VAR 
	i :INT;
END_VAR
// enable/disenable joint5
IF i_setupArm.jnt5AdjustDir = 0 THEN
	m_jntEnableFlag[5] := 0;
	m_cmdJntPos[5]:=i_setupArm.curJntPos[5];
	m_jnt5EnableTime:=0;
	m_cmdJntVel[5]:=0;
	RETURN;
ELSE
	m_jntEnableFlag[5] := 1;
	m_jnt5EnableTime := m_jnt5EnableTime + g_setupArmCtrlCycleTime;
END_IF

// update command position
IF m_jnt5EnableTime>m_jnt5AdjustWaitTime THEN
	m_cmdJntVel[5]:=m_cmdJntVel[5] + i_setupArm.jnt5AdjustDir * m_jnt5MaxAdjustAcc * g_setupArmCtrlCycleTime;
	m_cmdJntVel[5]:=LIMIT(-m_jnt5MaxAdjustVel, m_cmdJntVel[5], m_jnt5MaxAdjustVel);
	
	// joint limit
	IF (m_cmdJntPos[5] > GVL_SetupMotorParameters.g_maxJntPos[i_setupArm.armIdx, 5] AND m_cmdJntVel[5]>0) OR (m_cmdJntPos[5] < GVL_SetupMotorParameters.g_minJntPos[i_setupArm.armIdx, 5] AND m_cmdJntVel[5]<0)  THEN
		m_cmdJntVel[5] := 0;
	END_IF
	
	m_cmdJntPos[5]:= m_cmdJntPos[5] + m_cmdJntVel[5] * g_setupArmCtrlCycleTime;
END_IF
END_METHOD

// override this function in each exact controller
METHOD PROTECTED calcCmdJntTrq : BOOL
VAR_IN_OUT CONSTANT
	i_setupArm	:FB_SetupArm;
END_VAR
VAR
	i:INT;
	vel :LREAL;
	scale:LREAL;
	ratio:LREAL;
END_VAR
// set joint torque to zero in default
m_cmdJntTrq := g_zeroVec5d;

//enable/diable  joint1-4
IF NOT(i_setupArm.manualAdjustOn) THEN
	FOR i:=1 TO 4 DO
		m_jntEnableFlag[i] := 0;
		m_jntOPMode[i]:=DriverOPMode_Pos;
	END_FOR
	RETURN;
ELSE
	FOR i:=1 TO 4 DO
		m_jntEnableFlag[i] := 1;
		m_jntOPMode[i]:=DriverOPMode_Trq;
		m_cmdJntPos[i] := i_setupArm.curJntPos[i];
	END_FOR
END_IF

// friction scale
vel:=ABS(i_setupArm.curJntVel[3]);
IF vel < m_jnt3FrictionCompVelLow THEN
	m_frictionScale := m_frictionScaleLow * vel/m_jnt3FrictionCompVelLow ;
ELSIF  vel > m_jnt3FrictionCompVelLow AND vel  < m_jnt3FrictionCompVelMiddle THEN
	ratio:= (vel-m_jnt3FrictionCompVelLow)/(m_jnt3FrictionCompVelMiddle-m_jnt3FrictionCompVelLow);
	m_frictionScale :=m_frictionScaleLow+ratio * (m_frictionScaleMiddle-m_frictionScaleLow);
ELSIF  vel > m_jnt3FrictionCompVelMiddle AND vel  < m_jnt3FrictionCompVelHigh THEN
	ratio:= (vel-m_jnt3FrictionCompVelMiddle)/(m_jnt3FrictionCompVelHigh-m_jnt3FrictionCompVelMiddle);
	m_frictionScale :=m_frictionScaleMiddle+ratio * (m_frictionScaleHigh-m_frictionScaleMiddle);
ELSIF  vel > m_jnt3FrictionCompVelHigh THEN
	m_frictionScale := m_frictionScaleHigh;
END_IF

// add friction compensation
m_frictionScale := LIMIT(0, m_frictionScale, 1);
m_cmdJntTrq[3]:= m_frictionScale * sign(i_setupArm.curJntVel[3])*jnt3Friction(i_setupArm.armIdx, i_setupArm.curJntPos[3]);
END_METHOD

METHOD PUBLIC init : BOOL
VAR_IN_OUT CONSTANT
	i_setupArm	:FB_SetupArm;
END_VAR
VAR_IN_OUT 
	r_setupArmCtrlCmd :ST_SetupArmCtrlCmds;
END_VAR
SUPER^.Init(i_setupArm,r_setupArmCtrlCmd);
m_jnt5EnableTime :=0;
END_METHOD

METHOD PROTECTED jnt3Friction : Lreal
VAR_INPUT
	i_armIdx:INT;
	i_jnt3Pos :LREAL;
END_VAR

VAR
	q:LREAL;
END_VAR
q := LIMIT(GVL_SetupArmDynamics.g_setupJnt3GravityPosRange[i_armIdx,1], i_jnt3Pos, GVL_SetupArmDynamics.g_setupJnt3GravityPosRange[i_armIdx,2]);
jnt3Friction:=GVL_SetupArmDynamics.g_setupJnt3FrictionParams[i_armIdx,1]*EXPT(q,3)+GVL_SetupArmDynamics.g_setupJnt3FrictionParams[i_armIdx,2]*EXPT(q,2)+
				GVL_SetupArmDynamics.g_setupJnt3FrictionParams[i_armIdx,3]*q+GVL_SetupArmDynamics.g_setupJnt3FrictionParams[i_armIdx,4];
END_METHOD

END_FUNCTION_BLOCK

// ---- FBs_SlaveControllers/FB_SlaveCtrlInstruInvasion.TcPOU
// Brief: Slave Arm Adjust
FUNCTION_BLOCK PUBLIC FB_SlaveCtrlInstruInvasion EXTENDS FB_SlaveArmCtrlBase
VAR_INPUT
END_VAR
VAR_OUTPUT
END_VAR
VAR
	// invasion buffer
	m_instruInvasionDepthSafetyBuffer :LREAL:= 0.01;
		
	// max damping when reaching invasion depth
	m_maxDamp :LREAL :=500;
	
	// current distance form target invasion depth 
	m_invasionDis :LREAL :=0;
	
	// distance threshold from target depth to start enable damp
	m_dampDisThres :LREAL :=0.03;
	
END_VAR

// override this function in each exact controller
METHOD PROTECTED calcCmdJntPos : BOOL
VAR_IN_OUT CONSTANT
	i_endoscopePose : ST_Frame;
	i_masterStatus :ST_MasterStatus;
	i_setupStatus: ST_SetupStatus;
	i_slaveArm :FB_SlaveArm;
END_VAR

VAR 
	curInstruDepth:LREAL;
END_VAR
m_cmdJntPos[3]:=i_slaveArm.curJntPos[3];
// compute current instrument depth
curInstruDepth := i_slaveArm.curJntPos[3]-i_slaveArm.instrument.kinematicParameters.m_rodLength-i_slaveArm.instrument.kinematicParameters.m_headLength
						- i_slaveArm.instrument.kinematicParameters.m_fingerLength-m_instruInvasionDepthSafetyBuffer;

m_invasionDis:=curInstruDepth-i_slaveArm.m_instruInvasionDepth;
						
m_isFinished := curInstruDepth<= i_slaveArm.m_instruInvasionDepth;
END_METHOD

// override this function in each exact controller
METHOD PROTECTED calcCmdJntTrq : BOOL
VAR_IN_OUT CONSTANT
	i_endoscopePose : ST_Frame;
	i_masterStatus :ST_MasterStatus;
	i_setupStatus: ST_SetupStatus;
	i_slaveArm :FB_SlaveArm;
END_VAR
VAR
	dampScale :lreal ;
END_VAR
// set joint torque to zero in default
m_cmdJntTrq := g_zeroVec8d;

dampScale  :=LIMIT(0, 1-m_invasionDis/m_dampDisThres,1);
m_cmdJntTrq[3]:= -dampScale * m_maxDamp * i_slaveArm.curJntVel[3];
END_METHOD

METHOD PUBLIC init : BOOL
VAR_IN_OUT CONSTANT
	i_slaveArm	:FB_SlaveArm;
END_VAR
VAR_IN_OUT 
	r_slaveArmCtrlCmd :ST_SlaveArmCtrlCmds;
END_VAR
// check if to hold the command joint position unchanged
m_holdLastCmds := checkToHoldLastCmds(i_slaveArm);

//init
SUPER^.Init(i_slaveArm,r_slaveArmCtrlCmd);
m_invasionDis:=m_dampDisThres;

// only joint 3 is allowed to be pushed
m_jntOPMode := g_slaveAllPosMode;
m_jntOPMode[3]:=DriverOPMode_Trq;

// update commands to arm
copyCmds(r_slaveArmCtrlCmd);
END_METHOD

END_FUNCTION_BLOCK

// ---- FBs_SlaveControllers/FB_SlaveCtrlInstruCali.TcPOU
// Brief: Mounting Instrument
FUNCTION_BLOCK PUBLIC FB_SlaveCtrlInstruCali EXTENDS FB_SlaveArmCtrlBase
VAR
	// mount motion planning
	m_jntOTG :ARRAY[1..8] OF FB_secOrdTrajFilter;
	m_instruMountVel :LREAL := 2*PI;
	m_instruMountAcc :LREAL := 4*PI;
	
	// 	cali status
	m_rollJntCaliStatus :INT := 0;
	m_pitchJntCaliStatus :INT := 0;
	m_yawJntCaliStatus :INT := 0;
	
	// flag if zero position is written to CoE
	m_zeroPosWritten :BOOL;
	
	// joint current threshold which indicate panel is buckled with instrument
	m_maxJntCurrent :LREAL := 100;
	
	// joint current threshold which indicate finger closed
	m_fingerCloseCurrent :LREAL := 50;
	
	// joint position at limits
	m_jntLimitPos1, m_jntLimitPos2, m_jntCaliPos :LREAL;
	m_jntLimitPos3, m_jntLimitPos4 :LREAL;

	// flag if joint is mounted
	m_jointMounted :ARRAY[1..8] OF BOOL := [5(FALSE)];
	
	// instrument mount motion range
	m_mountMotionAng :LREAL :=pi;
	
	// command mount motion
	m_targetMountPos :Vec8d;
	
	// instrument zero position
	m_instruZeroPosition :Vec5d;
	
END_VAR

// override this function in each exact controller
METHOD PROTECTED calcCmdJntPos : BOOL
VAR_IN_OUT CONSTANT
	i_endoscopePose : ST_Frame;
	i_masterStatus :ST_MasterStatus;
	i_setupStatus: ST_SetupStatus;
	i_slaveArm :FB_SlaveArm;
END_VAR

VAR 
	i :INT;
END_VAR
// retur directly if instrument/endoscope is not readed
IF NOT i_slaveArm.instrument.onChipData.m_InstruReadSucceed THEN
	m_rollJntCaliStatus :=0;
	m_pitchJntCaliStatus :=0;
	m_yawJntCaliStatus :=0;
	m_zeroPosWritten :=FALSE;
	FOR i:=4 TO 8 DO
		m_jointMounted[i]:=FALSE;
	END_FOR
	return;
END_IF

// write zero position to CoE
IF m_yawJntCaliStatus = -1 THEN
	IF   NOT m_zeroPosWritten THEN
		m_zeroPosWritten := i_slaveArm.instrument.writeZeroPosToChip(m_instruZeroPosition[1],m_instruZeroPosition[2],m_instruZeroPosition[3]);
	END_IF
	RETURN;
END_IF;

// move joint to zero position
IF m_rollJntCaliStatus <> -1 THEN
	rollJntCali(i_slaveArm);
ELSIF m_pitchJntCaliStatus <> -1 THEN
	pitchJntCali(i_slaveArm);
ELSIF m_yawJntCaliStatus <> -1 THEN
	IF  i_slaveArm.instrument.m_isSingleFinger THEN
		yawJntCali_finger(i_slaveArm);
	ELSE
		yawJntCali_gripper(i_slaveArm);
	END_IF

END_IF

IF m_yawJntCaliStatus = -1 THEN
	FOR  i:=1 TO  5 DO
		m_instruZeroPosition[i]:=i_slaveArm.linkSingle[i+3];
	END_FOR
END_IF
END_METHOD

METHOD PUBLIC init : BOOL
VAR_IN_OUT CONSTANT
	i_slaveArm	:FB_SlaveArm;
END_VAR
VAR_IN_OUT 
	r_slaveArmCtrlCmd :ST_SlaveArmCtrlCmds;
END_VAR

VAR
	i : INT;
END_VAR
// check if to hold the command joint position unchanged
m_holdLastCmds := checkToHoldLastCmds(i_slaveArm);

SUPER^.Init(i_slaveArm,r_slaveArmCtrlCmd);
m_jntOPMode[4] := DriverOPMode_PosTrq;
m_jntOPMode[5] := DriverOPMode_PosTrq;
m_jntOPMode[6] := DriverOPMode_PosTrq;
m_jntOPMode[7] := DriverOPMode_PosTrq;
m_jntOPMode[8] := DriverOPMode_PosTrq;

FOR i:=4 TO 8 DO
	m_targetMountPos[i]:=m_cmdJntPos[i];
	m_jntOTG[i].init(m_targetMountPos[i], 0,m_instruMountVel, m_instruMountAcc, g_slaveArmCtrlCycleTime);
	m_jointMounted[i]:=FALSE;
END_FOR

m_rollJntCaliStatus :=0;
m_pitchJntCaliStatus :=0;
m_yawJntCaliStatus :=0;
m_zeroPosWritten := false;

// update commands to arm
copyCmds(r_slaveArmCtrlCmd);
END_METHOD

METHOD pitchJntCali : BOOL
VAR_IN_OUT CONSTANT
	i_slaveArm :FB_SlaveArm;
END_VAR

VAR 
	i :INT;
	curJntPos :Vec8d;
	jntIdx :INT;
END_VAR
jntIdx:=6;
curJntPos := i_slaveArm.curJntPos;

CASE m_pitchJntCaliStatus OF
	// rotate clockwise
	0:
		m_targetMountPos[jntIdx]:=curJntPos[jntIdx]+m_mountMotionAng;
	
		//buckle joint
		IF i_slaveArm.filtJntCurrent[jntIdx]> m_maxJntCurrent THEN 
			m_jntLimitPos1 := curJntPos[jntIdx];
			m_targetMountPos[jntIdx]:=curJntPos[jntIdx];
			m_jntOTG[jntIdx].init(m_targetMountPos[jntIdx], 0,m_instruMountVel, m_instruMountAcc, g_slaveArmCtrlCycleTime);
			m_pitchJntCaliStatus := 1;
		END_IF
		
	// rotate anticlockwise
	1:
		m_targetMountPos[jntIdx]:=curJntPos[jntIdx]-m_mountMotionAng;
	
		//buckle  joint
		IF i_slaveArm.filtJntCurrent[jntIdx]<- m_maxJntCurrent THEN 
			m_jntLimitPos2 := curJntPos[jntIdx];
			m_targetMountPos[jntIdx]:=curJntPos[jntIdx];
			m_jntOTG[jntIdx].init(m_targetMountPos[jntIdx], 0,m_instruMountVel, m_instruMountAcc, g_slaveArmCtrlCycleTime);
			m_pitchJntCaliStatus := 2;
		END_IF
	
	2:// calculate center/calibarted position
		m_targetMountPos[jntIdx] :=  (m_jntLimitPos1 + m_jntLimitPos2)/2;
		m_pitchJntCaliStatus := 3;

	3:
		IF ABS(m_targetMountPos[jntIdx]-curJntPos[jntIdx]) <GVL_SlaveControlParameters.g_jntCtrlAngTolHigh  THEN
			m_pitchJntCaliStatus := -1;
		END_IF
		
END_CASE

// traj plan
m_jntOTG[jntIdx].run(m_targetMountPos[jntIdx],0.0, o_cmdAcc=>m_cmdJntAcc[jntIdx],o_cmdVel=>m_cmdJntVel[jntIdx],o_cmdPos=>m_cmdJntPos[jntIdx]);
END_METHOD

METHOD rollJntCali : BOOL
VAR_IN_OUT CONSTANT
	i_slaveArm :FB_SlaveArm;
END_VAR

VAR 
	i :INT;
	curJntPos :Vec8d;
	jntIdx :INT;
END_VAR
jntIdx:=7;
curJntPos := i_slaveArm.curJntPos;

CASE m_rollJntCaliStatus OF
	// rotate clockwise
	0:
		m_targetMountPos[jntIdx]:=curJntPos[jntIdx]+m_mountMotionAng;
	
		//buckle  joint
		IF i_slaveArm.filtJntCurrent[jntIdx]> m_maxJntCurrent THEN 
			m_jntLimitPos1 := curJntPos[jntIdx];
			m_targetMountPos[jntIdx]:=curJntPos[jntIdx];
			m_jntOTG[jntIdx].init(m_targetMountPos[jntIdx], 0,m_instruMountVel, m_instruMountAcc, g_slaveArmCtrlCycleTime);
			m_rollJntCaliStatus := 1;
		END_IF
		
	// rotate anticlockwise
	1:
		m_targetMountPos[jntIdx]:=curJntPos[jntIdx]-m_mountMotionAng;
	
		//buckle  joint
		IF i_slaveArm.filtJntCurrent[jntIdx]<- m_maxJntCurrent THEN 
			m_jntLimitPos2 := curJntPos[jntIdx];
			m_targetMountPos[jntIdx]:=curJntPos[jntIdx];
			m_jntOTG[jntIdx].init(m_targetMountPos[jntIdx], 0,m_instruMountVel, m_instruMountAcc, g_slaveArmCtrlCycleTime);
			m_rollJntCaliStatus := 2;
		END_IF
	
	2:// calculate center/calibarted positio
		m_targetMountPos[jntIdx] :=  (m_jntLimitPos1 + m_jntLimitPos2)/2;
		m_rollJntCaliStatus := 3;

	3:
		IF ABS(m_targetMountPos[jntIdx]-curJntPos[jntIdx]) <GVL_SlaveControlParameters.g_jntCtrlAngTolHigh  THEN
			m_rollJntCaliStatus := -1;
		END_IF
		
END_CASE

// traj plan
m_jntOTG[jntIdx].run(m_targetMountPos[jntIdx],0.0, o_cmdAcc=>m_cmdJntAcc[jntIdx],o_cmdVel=>m_cmdJntVel[jntIdx],o_cmdPos=>m_cmdJntPos[jntIdx]);
END_METHOD

METHOD yawJntCali_finger : BOOL
VAR_IN_OUT CONSTANT
	i_slaveArm :FB_SlaveArm;
END_VAR

VAR 
	i :INT;
	curJntPos :Vec8d;
	jntIdx :INT;
END_VAR
jntIdx:=5;
curJntPos := i_slaveArm.curJntPos;

CASE m_yawJntCaliStatus OF
	// rotate clockwise
	0:
		m_targetMountPos[jntIdx]:=curJntPos[jntIdx]+m_mountMotionAng;
	
		//buckle  joint
		IF i_slaveArm.filtJntCurrent[jntIdx]> m_maxJntCurrent THEN 
			m_jntLimitPos1 := curJntPos[jntIdx];
			m_targetMountPos[jntIdx]:=curJntPos[jntIdx];
			m_jntOTG[jntIdx].init(m_targetMountPos[jntIdx], 0,m_instruMountVel, m_instruMountAcc, g_slaveArmCtrlCycleTime);
			m_yawJntCaliStatus := 1;
		END_IF
		
	// rotate anticlockwise
	1:
		m_targetMountPos[jntIdx]:=curJntPos[jntIdx]-m_mountMotionAng;
	
		//buckle  joint
		IF i_slaveArm.filtJntCurrent[jntIdx]<- m_maxJntCurrent THEN 
			m_jntLimitPos2 := curJntPos[jntIdx];
			m_targetMountPos[jntIdx]:=curJntPos[jntIdx];
			m_jntOTG[jntIdx].init(m_targetMountPos[jntIdx], 0,m_instruMountVel, m_instruMountAcc, g_slaveArmCtrlCycleTime);
			m_yawJntCaliStatus := 2;
		END_IF
	
	2:// calculate center/calibarted positio
		m_targetMountPos[jntIdx] :=  (m_jntLimitPos1 + m_jntLimitPos2)/2;
		m_yawJntCaliStatus := 3;

	3:
		IF ABS(m_targetMountPos[jntIdx]-curJntPos[jntIdx]) <GVL_SlaveControlParameters.g_jntCtrlAngTolHigh  THEN
			m_yawJntCaliStatus := -1;
		END_IF
		
END_CASE

// traj plan
m_jntOTG[jntIdx].run(m_targetMountPos[jntIdx],0.0, o_cmdAcc=>m_cmdJntAcc[jntIdx],o_cmdVel=>m_cmdJntVel[jntIdx],o_cmdPos=>m_cmdJntPos[jntIdx]);
END_METHOD

METHOD yawJntCali_gripper : BOOL
VAR_IN_OUT CONSTANT
	i_slaveArm :FB_SlaveArm;
END_VAR

VAR 
	i :INT;
	curJntPos :Vec8d;
	jntRange:LREAL;
	jntIdx :INT;
END_VAR
curJntPos := i_slaveArm.curJntPos;

CASE m_yawJntCaliStatus OF
	// roll clockwise
	0:
		//buckle panel with instrument
		// check if buckled 
		IF i_slaveArm.filtJntCurrent[4]<- m_maxJntCurrent THEN 
			m_jointMounted[4]:=TRUE;
			m_targetMountPos[4]:=curJntPos[4];
			m_jntOTG[4].init(m_targetMountPos[4], 0,m_instruMountVel, m_instruMountAcc, g_slaveArmCtrlCycleTime);
		END_IF
		IF i_slaveArm.filtJntCurrent[5]> m_maxJntCurrent THEN 
			m_jointMounted[5]:=TRUE;
			m_targetMountPos[5]:=curJntPos[5];
			m_jntOTG[5].init(m_targetMountPos[5], 0,m_instruMountVel, m_instruMountAcc, g_slaveArmCtrlCycleTime);
		END_IF
		
		// set target joint position
		IF FALSE = m_jointMounted[4] THEN
			m_targetMountPos[4]:=curJntPos[4]-m_mountMotionAng;
		END_IF
		IF FALSE = m_jointMounted[5] THEN
			m_targetMountPos[5]:=curJntPos[5]+m_mountMotionAng;
		END_IF

		IF m_jointMounted[4] AND m_jointMounted[5] THEN
			m_jntLimitPos1 := curJntPos[4];
			m_jntLimitPos2 := curJntPos[5];
			m_yawJntCaliStatus := 1;
			m_jointMounted[4]:=FALSE;
			m_jointMounted[5]:=FALSE;
		END_IF

	// roll anticlockwise
	1:
		IF i_slaveArm.filtJntCurrent[4]> m_maxJntCurrent THEN 
			m_jointMounted[4]:=TRUE;
			m_targetMountPos[4]:=curJntPos[4];
			m_jntOTG[4].init(m_targetMountPos[4], 0,m_instruMountVel, m_instruMountAcc, g_slaveArmCtrlCycleTime);
		END_IF
		IF i_slaveArm.filtJntCurrent[5]<- m_maxJntCurrent THEN 
			m_jointMounted[5]:=TRUE;
			m_targetMountPos[5]:=curJntPos[5];
			m_jntOTG[5].init(m_targetMountPos[5], 0,m_instruMountVel, m_instruMountAcc, g_slaveArmCtrlCycleTime);
		END_IF
		
		// set target joint position
		IF FALSE = m_jointMounted[4] THEN
			m_targetMountPos[4]:=curJntPos[4]+m_mountMotionAng;
		END_IF
		IF FALSE = m_jointMounted[5] THEN
			m_targetMountPos[5]:=curJntPos[5]-m_mountMotionAng;
		END_IF
		
		IF m_jointMounted[4] AND m_jointMounted[5] THEN
			m_jntLimitPos3 := curJntPos[4];
			m_jntLimitPos4 := curJntPos[5];
			m_yawJntCaliStatus :=2;
			m_jointMounted[4]:=FALSE;
			m_jointMounted[5]:=FALSE;
		END_IF
		
	2:// calculate center/calibarted position
		m_targetMountPos[4] := (m_jntLimitPos1 + m_jntLimitPos3)/2;
		m_targetMountPos[5] := (m_jntLimitPos2 + m_jntLimitPos4)/2;
		m_yawJntCaliStatus := 3;

	3:
		IF ABS(m_targetMountPos[4]-curJntPos[4]) <GVL_SlaveControlParameters.g_jntCtrlAngTolHigh  AND
			ABS(m_targetMountPos[5]-curJntPos[5]) <GVL_SlaveControlParameters.g_jntCtrlAngTolHigh  THEN
			m_yawJntCaliStatus := 4;
		END_IF
		
	// close finger
	4:
		//buckle panel with instrument
		FOR i:=4 TO 5 DO
			// check if buckled 
			IF i_slaveArm.filtJntCurrent[i]> m_fingerCloseCurrent THEN 
				m_jointMounted[i]:=TRUE;
				m_targetMountPos[i]:=curJntPos[i];
				m_jntOTG[i].init(m_targetMountPos[i], 0,m_instruMountVel, m_instruMountAcc, g_slaveArmCtrlCycleTime);
			END_IF
			
			// set target joint position
			IF FALSE = m_jointMounted[i] THEN
				m_targetMountPos[i]:=curJntPos[i]+m_mountMotionAng;
			END_IF
		END_FOR
		
		IF m_jointMounted[4] AND m_jointMounted[5] THEN
			m_yawJntCaliStatus := -1;
		END_IF
END_CASE

// traj plan
m_jntOTG[4].run(m_targetMountPos[4],0.0, o_cmdAcc=>m_cmdJntAcc[4],o_cmdVel=>m_cmdJntVel[4],o_cmdPos=>m_cmdJntPos[4]);
m_jntOTG[5].run(m_targetMountPos[5],0.0, o_cmdAcc=>m_cmdJntAcc[5],o_cmdVel=>m_cmdJntVel[5],o_cmdPos=>m_cmdJntPos[5]);
END_METHOD

END_FUNCTION_BLOCK

// ---- FBs_SlaveControllers/FB_SlaveCtrlError.TcPOU
// Brief: Slave Arm Error Hold
FUNCTION_BLOCK PUBLIC FB_SlaveCtrlError EXTENDS FB_SlaveArmCtrlBase
VAR_INPUT
END_VAR
VAR_OUTPUT
END_VAR
VAR
END_VAR

// override this function in each exact controller
METHOD PROTECTED calcCmdJntPos : BOOL
VAR_IN_OUT CONSTANT
	// endoscope pose in cart coordinate
	i_endoscopePose : ST_Frame;
	
	// master arm data
	i_masterStatus :ST_MasterStatus;
	
	// setup arm data
	i_setupStatus: ST_SetupStatus;
	
	// slave arm data
	i_slaveArm :FB_SlaveArm;
END_VAR
m_cmdJntPos := i_slaveArm.curJntPos;
END_METHOD

// override this function in each exact controller
// NOTICE: set joint control mode here, and do some initialization if needed
METHOD PUBLIC init : BOOL
VAR_IN_OUT CONSTANT
	i_slaveArm	:FB_SlaveArm;
END_VAR
VAR_IN_OUT 
	r_slaveArmCtrlCmd :ST_SlaveArmCtrlCmds;
END_VAR


VAR
	i:INT;
END_VAR
SUPER^.Init(i_slaveArm,r_slaveArmCtrlCmd);

// disable all joints
 m_jntEnableFlag :=g_zeroVec8i;
 
 // update commands to arm
copyCmds(r_slaveArmCtrlCmd);
END_METHOD

END_FUNCTION_BLOCK

// ---- FBs_SlaveControllers/FB_SlaveCtrlMountInstru.TcPOU
// Brief: Mounting Instrument
FUNCTION_BLOCK PUBLIC FB_SlaveCtrlMountInstru EXTENDS FB_SlaveArmCtrlBase
VAR
	// mount status
	m_instruMountStatus :INT := 0;
	m_scopeMountStatus :INT := 0;
	m_ultrasoundMountStatus :INT :=0 ;
	
	// flag if joint is mounted
	m_jointMounted :ARRAY[1..5] OF BOOL := [5(FALSE)];
	
	// instrument mount motion range
	m_mountMotionAng :Vec5d :=[5(pi)];
	
	// instrument mount direction
	m_mountDir :Vec5i :=[1, 1, 1, 1, 1];
	
	// mount motion planning
	m_jntOTG :ARRAY[1..5] OF FB_secOrdTrajFilter;
	m_instruMountVel :LREAL := 4*PI;
	m_instruMountAcc :LREAL := 8*PI;
	
	//Joint 4 half-range angle of instrument
	m_instruJnt4HalfRangeAng :LREAL := 323*g_deg2Rad;
	
	// joint current threshold which indicate panel is buckled with instrument
	m_maxJntCurrent :Vec5d := [150, 150, 150, 180, 180];
	
	// command mount motion
	m_targetMountPos :Vec8d;
	
	// instrument zero position
	m_instruZeroDeviation :Vec5d;
	
	//ultrasound knife Reduce the current rotation Angle  J3
	m_ultraKnifeRotaAngleJ3 :LREAL := 3*g_deg2Rad;
	
	// joint position error
	m_jntPosErr :Vec5d;
	
	// endoscope motion angle to original position
	m_scopeJnt4CenterMotionAng :LREAL :=175*g_deg2Rad;
	m_scopeJnt5CenterMotionAng :LREAL :=150*g_deg2Rad;
	
END_VAR

// override this function in each exact controller
METHOD PROTECTED calcCmdJntPos : BOOL
VAR_IN_OUT CONSTANT
	i_endoscopePose : ST_Frame;
	i_masterStatus :ST_MasterStatus;
	i_setupStatus: ST_SetupStatus;
	i_slaveArm :FB_SlaveArm;
END_VAR

VAR 
END_VAR
// return directly if instrument/endoscope is not readed
IF i_slaveArm.instrument.onChipData.m_Error THEN
	return;
END_IF

IF i_slaveArm.instrument.onChipData.m_InstruReadSucceed AND InstruType_endoscope = i_slaveArm.instrument.m_instruType THEN
	mountEndoscope(i_slaveArm);
ELSIF i_slaveArm.instrument.onChipData.m_InstruReadSucceed AND InstruType_UltrasoundKnife = i_slaveArm.instrument.m_instruType THEN
	mountUltraKnife(i_slaveArm);
ELSE
	mountInstrument(i_slaveArm);
END_IF
END_METHOD

METHOD PUBLIC init : BOOL
VAR_IN_OUT CONSTANT
	i_slaveArm	:FB_SlaveArm;
END_VAR
VAR_IN_OUT 
	r_slaveArmCtrlCmd :ST_SlaveArmCtrlCmds;
END_VAR

VAR
	i : INT;
END_VAR
// check if to hold the command joint position unchanged
m_holdLastCmds := checkToHoldLastCmds(i_slaveArm);

SUPER^.Init(i_slaveArm,r_slaveArmCtrlCmd);
m_jntOPMode[4] := DriverOPMode_PosTrq;
m_jntOPMode[5] := DriverOPMode_PosTrq;
m_jntOPMode[6] := DriverOPMode_PosTrq;
m_jntOPMode[7] := DriverOPMode_PosTrq;
m_jntOPMode[8] := DriverOPMode_PosTrq;

FOR i:=1 TO 5 DO
	m_targetMountPos[i+3]:=m_cmdJntPos[i+3];
	m_jntOTG[i].init(m_targetMountPos[i+3], 0,m_instruMountVel, m_instruMountAcc, g_slaveArmCtrlCycleTime);
	m_jointMounted[i]:=FALSE;
END_FOR

m_instruMountStatus:=0;
m_scopeMountStatus:=0;
m_ultrasoundMountStatus:=0;

// update commands to arm
copyCmds(r_slaveArmCtrlCmd);
END_METHOD

METHOD mountEndoscope : BOOL
VAR_IN_OUT CONSTANT
	i_slaveArm :FB_SlaveArm;
END_VAR

VAR 
	i :INT;
	curJntPos :Vec8d;
END_VAR
curJntPos := i_slaveArm.curJntPos;

CASE m_scopeMountStatus OF
	//fix scope lock joint(joint 7)
	0:
		// other joints stay still
		FOR i:=1 TO 3 DO
			m_jointMounted[i] := TRUE;
			m_targetMountPos[i+3]:=curJntPos[i+3];
			m_jntOTG[i].init(m_targetMountPos[i+3], 0,m_instruMountVel, m_instruMountAcc, g_slaveArmCtrlCycleTime);
		END_FOR
	
		// check if buckled
		m_jointMounted[4]:=FALSE; 
		m_jointMounted[5]:=FALSE; 
		IF ABS(i_slaveArm.filtJntCurrent[7])> m_maxJntCurrent[4] THEN 
			m_jointMounted[4]:=TRUE;
			m_targetMountPos[7]:=curJntPos[7];
			m_jntOTG[4].init(m_targetMountPos[7], 0,m_instruMountVel, m_instruMountAcc, g_slaveArmCtrlCycleTime);
			m_scopeMountStatus:=1;
		ELSE
			m_targetMountPos[7]:=curJntPos[7]+m_mountMotionAng[4];
		END_IF

	1: // buckle scope rotate joint (joint 8)
		m_jointMounted[5]:=FALSE; 
		IF ABS(i_slaveArm.filtJntCurrent[8])> m_maxJntCurrent[5] THEN 
			m_jointMounted[5]:=TRUE;
			m_targetMountPos[8]:=curJntPos[8];
			m_jntOTG[5].init(m_targetMountPos[8], 0,m_instruMountVel, m_instruMountAcc, g_slaveArmCtrlCycleTime);
			m_scopeMountStatus:=2;
		ELSE
			m_targetMountPos[8]:=curJntPos[8]+m_mountMotionAng[5];
		END_IF
	

	2:// move back to zero position
		m_targetMountPos[7]:= curJntPos[7]-m_scopeJnt4CenterMotionAng;
		m_targetMountPos[8]:= curJntPos[8]-m_scopeJnt5CenterMotionAng;
		m_scopeMountStatus :=3;
		
		
	3:
		IF ABS(m_targetMountPos[7]-curJntPos[7]) <GVL_SlaveControlParameters.g_jntCtrlAngTolHigh AND 
				ABS(m_targetMountPos[8]-curJntPos[8]) <GVL_SlaveControlParameters.g_jntCtrlAngTolHigh THEN
			m_isFinished := TRUE;
		END_IF
		
END_CASE

// traj plan
FOR i:=1 TO 5 DO
	m_jntOTG[i].run(m_targetMountPos[i+3],0.0, o_cmdAcc=>m_cmdJntAcc[3+i],o_cmdVel=>m_cmdJntVel[3+i],o_cmdPos=>m_cmdJntPos[i+3]);
END_FOR
END_METHOD

METHOD mountInstrument : BOOL
VAR_IN_OUT CONSTANT
	i_slaveArm :FB_SlaveArm;
END_VAR

VAR 
	i :INT;
	curJntPos :Vec8d;
END_VAR
curJntPos := i_slaveArm.curJntPos;

// joint4 stay still if instrument has only on finger
IF i_slaveArm.instrument.m_isSingleFinger THEN
	m_jointMounted[1]:=TRUE;
END_IF

CASE m_instruMountStatus OF
	// To lock panel with instrument
	0:
		//buckle panel with instrument
		FOR i:=1 TO 4 DO
			// check if buckled 
			IF ABS(i_slaveArm.filtJntCurrent[i+3])> m_maxJntCurrent[i] THEN 
				m_jointMounted[i]:=TRUE;
				m_targetMountPos[i+3]:=curJntPos[i+3];
				m_jntOTG[i].init(m_targetMountPos[i+3], 0,m_instruMountVel, m_instruMountAcc, g_slaveArmCtrlCycleTime);
			END_IF
			
			// set target joint position
			IF FALSE = m_jointMounted[i] THEN
				m_targetMountPos[i+3]:=curJntPos[i+3]-m_mountMotionAng[i];
			END_IF
		END_FOR
		
		
		// check transition condition
		IF (m_jointMounted[1] AND m_jointMounted[2] AND m_jointMounted[3] AND m_jointMounted[4])  THEN
			IF i_slaveArm.instrument.onChipData.m_InstruReadSucceed THEN//Check whether the data is read successfully
				m_instruMountStatus:=1;
			END_IF
		END_IF
	
	1:// calculation deviates from the instrument zero position
		FOR i:=1 TO 4 DO
			m_instruZeroDeviation[i] :=  i_slaveArm.linkSingle[i+3] - i_slaveArm.instrument.onChipData.m_InstruPos[i];
		END_FOR
		m_instruMountStatus :=2;
	
	
	2:// move back to zero position
		FOR i:=1 TO 3 DO//J1-3
			IF m_instruZeroDeviation[i]>pi THEN
				m_instruZeroDeviation[i] := m_instruZeroDeviation[i] - 2*PI;
			ELSIF m_instruZeroDeviation[i]<-pi THEN
				m_instruZeroDeviation[i] := m_instruZeroDeviation[i] + 2*PI;
			END_IF
		END_FOR
		
		//joint4
		IF m_instruZeroDeviation[4]>0 AND m_instruZeroDeviation[4] < pi THEN
			m_instruZeroDeviation[4] := m_instruZeroDeviation[4] - 2*pi;
		ELSIF m_instruZeroDeviation[4]<0 AND m_instruZeroDeviation[4] > -pi THEN
			m_instruZeroDeviation[4] := m_instruZeroDeviation[4] + 2*pi;
		END_IF
		
		// set target joint position
		FOR i:=1 TO 4 DO
			m_targetMountPos[i+3]:=curJntPos[i+3] - m_instruZeroDeviation[i];
		END_FOR
		m_instruMountStatus :=3;
		
		
	3:
		m_isFinished:=TRUE;
		FOR i:=1 TO 4 DO 
			m_jntPosErr[i]:=m_targetMountPos[i+3]-curJntPos[i+3];
			IF ABS(m_jntPosErr[i]) >GVL_SlaveControlParameters.g_jntCtrlAngTolHigh OR 
					ABS( i_slaveArm.linkSingle[i+3] - i_slaveArm.instrument.onChipData.m_InstruPos[i]) >5*g_deg2rad THEN
				m_isFinished := FALSE;
				EXIT;
			END_IF
		END_FOR
		
END_CASE

// traj plan
FOR i:=1 TO 4 DO
	m_jntOTG[i].run(m_targetMountPos[i+3],0.0, o_cmdAcc=>m_cmdJntAcc[3+i],o_cmdVel=>m_cmdJntVel[3+i],o_cmdPos=>m_cmdJntPos[i+3]);
END_FOR
END_METHOD

METHOD mountUltraKnife : BOOL
VAR_IN_OUT CONSTANT
	i_slaveArm :FB_SlaveArm;
END_VAR

VAR 
	i :INT;
	curJntPos :Vec8d;
END_VAR
curJntPos := i_slaveArm.curJntPos;

m_jointMounted[1]:=TRUE;
m_jointMounted[2]:=TRUE;


CASE m_ultrasoundMountStatus OF 
	// To lock panel with instrument
	0:
		//buckle panel with instrument
		FOR i:=3 TO 5 DO
			// check if buckled 
			IF ABS(i_slaveArm.filtJntCurrent[i+3])> m_maxJntCurrent[i] THEN 
				m_jointMounted[i]:=TRUE;
				m_targetMountPos[i+3]:=curJntPos[i+3];
				m_jntOTG[i].init(m_targetMountPos[i+3], 0,m_instruMountVel, m_instruMountAcc, g_slaveArmCtrlCycleTime);
			END_IF
			
			// set target joint position
			IF FALSE = m_jointMounted[i] THEN
				IF i = 5 THEN
					m_targetMountPos[i+3]:=curJntPos[i+3]+m_mountMotionAng[i];
				ELSE
					m_targetMountPos[i+3]:=curJntPos[i+3]-m_mountMotionAng[i];
				END_IF
				
			END_IF
		END_FOR

		// check transition condition
		IF ( m_jointMounted[3] AND m_jointMounted[4] AND m_jointMounted[5] )  THEN
			IF i_slaveArm.instrument.onChipData.m_InstruReadSucceed THEN//Check whether the data is read successfully
				m_ultrasoundMountStatus:=1;
			END_IF
		END_IF

	1:
		//m_jntOPMode[8] := DriverOPMode_Trq;
		// calculation deviates from the instrument zero position
		m_instruZeroDeviation[3] :=  m_ultraKnifeRotaAngleJ3;
		m_instruZeroDeviation[4] :=  i_slaveArm.linkSingle[7] - i_slaveArm.instrument.onChipData.m_InstruPos[4];
		m_ultrasoundMountStatus :=2;
		
	2:// move back to zero position
		//joint4
		IF m_instruZeroDeviation[4]>0 AND m_instruZeroDeviation[4] < pi THEN
			m_instruZeroDeviation[4] := m_instruZeroDeviation[4] - 2*pi;
		ELSIF m_instruZeroDeviation[4]<0 AND m_instruZeroDeviation[4] > -pi THEN
			m_instruZeroDeviation[4] := m_instruZeroDeviation[4] + 2*pi;
		END_IF
	
		// set target joint position
		m_targetMountPos[6]:=curJntPos[6] + m_instruZeroDeviation[3];
		m_targetMountPos[7]:=curJntPos[7] - m_instruZeroDeviation[4];
		m_targetMountPos[8]:=curJntPos[8] - m_instruZeroDeviation[4];

		m_ultrasoundMountStatus :=3;

	3:
		m_isFinished:=TRUE;
		FOR i:=3 TO 4 DO 
			m_jntPosErr[i]:=m_targetMountPos[i+3]-curJntPos[i+3];
			IF ABS(m_jntPosErr[i]) >GVL_SlaveControlParameters.g_jntCtrlAngTolHigh  THEN
				m_isFinished := FALSE;
				EXIT;
			END_IF
		END_FOR	

END_CASE


// traj plan
FOR i:=1 TO 5 DO
	m_jntOTG[i].run(m_targetMountPos[i+3],0.0, o_cmdAcc=>m_cmdJntAcc[3+i],o_cmdVel=>m_cmdJntVel[3+i],o_cmdPos=>m_cmdJntPos[i+3]);
END_FOR
END_METHOD

END_FUNCTION_BLOCK

// ---- FBs_SlaveControllers/FB_SlaveCtrlAdjust.TcPOU
// Brief: Slave Arm Adjust
FUNCTION_BLOCK PUBLIC FB_SlaveCtrlAdjust EXTENDS FB_SlaveArmCtrlBase
VAR_INPUT
END_VAR
VAR_OUTPUT
END_VAR
VAR
END_VAR

// override this function in each exact controller
METHOD PROTECTED calcCmdJntPos : BOOL
VAR_IN_OUT CONSTANT
	i_endoscopePose : ST_Frame;
	i_masterStatus :ST_MasterStatus;
	i_setupStatus: ST_SetupStatus;
	i_slaveArm :FB_SlaveArm;
END_VAR
m_cmdJntPos[1]:=i_slaveArm.curJntPos[1];
m_cmdJntPos[2]:=i_slaveArm.curJntPos[2];
m_cmdJntPos[3]:=i_slaveArm.curJntPos[3];
m_cmdJntPos[7]:=i_slaveArm.curJntPos[7];
m_cmdCartPose:=i_slaveArm.curCartPose;
END_METHOD

// override this function in each exact controller
METHOD PROTECTED calcCmdJntTrq : BOOL
VAR_IN_OUT CONSTANT
	i_endoscopePose : ST_Frame;
	i_masterStatus :ST_MasterStatus;
	i_setupStatus: ST_SetupStatus;
	i_slaveArm :FB_SlaveArm;
END_VAR
// set joint torque to zero in default
m_cmdJntTrq := g_zeroVec8d;
END_METHOD

METHOD PUBLIC init : BOOL
VAR_IN_OUT CONSTANT
	i_slaveArm	:FB_SlaveArm;
END_VAR
VAR_IN_OUT 
	r_slaveArmCtrlCmd :ST_SlaveArmCtrlCmds;
END_VAR
// check if to hold the command joint position unchanged
m_holdLastCmds := checkToHoldLastCmds(i_slaveArm);

//init
SUPER^.Init(i_slaveArm,r_slaveArmCtrlCmd);


// joint 1/2/3/7 run in torque mode
m_jntOPMode[1]:=DriverOPMode_Trq;
m_jntOPMode[2]:=DriverOPMode_Trq;
m_jntOPMode[3]:=DriverOPMode_Trq;
m_jntOPMode[4]:=DriverOPMode_PosTrq;
m_jntOPMode[5]:=DriverOPMode_PosTrq;
m_jntOPMode[6]:=DriverOPMode_PosTrq;
m_jntOPMode[7]:=DriverOPMode_Trq;
m_jntOPMode[8]:=DriverOPMode_PosTrq;

// update commands to arm
copyCmds(r_slaveArmCtrlCmd);
END_METHOD

END_FUNCTION_BLOCK

// ---- FBs_SlaveControllers/FB_SlaveCtrlGraCali.TcPOU
// Brief: Slave Arm Gravity Calibration
FUNCTION_BLOCK PUBLIC FB_SlaveCtrlGraCali EXTENDS FB_SlaveArmCtrlBase
VAR_INPUT
END_VAR
VAR_OUTPUT
END_VAR
VAR
// cali trajectory
	m_caliMotionSegs :INT :=3;
	m_graCaliTraj:ARRAY [1..3, 1..g_sJntNum] OF LREAL:=
		[-pi/6, -PI/2+pi/6, 0.5, 	5(0),
		 pi/6, 	-PI/2-pi/4, 0.3, 	5(0),
		 -pi/6, -PI/2+pi/6, 0.5, 	5(0)];
		 
	m_caliMaxjntVel:Vec8d:=[2(2.5*g_deg2Rad), 0.01, 5(2.5*g_deg2Rad)];
	m_caliMaxjntAcc:Vec8d:=[8(0.5)];
	m_caliMaxjntJerk:Vec8d:=[8(2.0)];
	
	m_caliTrajIdx: INT := 1;
	m_caliPlanner: ARRAY[1..3] OF FB_TrajMoveJ;
	
END_VAR

// override this function in each exact controller
METHOD PROTECTED calcCmdJntPos : BOOL
VAR_IN_OUT CONSTANT
	i_endoscopePose : ST_Frame;
	i_masterStatus :ST_MasterStatus;
	i_setupStatus: ST_SetupStatus;
	i_slaveArm :FB_SlaveArm;
END_VAR


VAR 
	i :INT;
	curJntVel :Vec8d;
END_VAR
// check if planner is ready
IF m_caliPlanner[m_caliTrajIdx].isGene = FALSE THEN
	calcCmdJntPos:=FALSE;
	RETURN;
END_IF

// traj plan
calcCmdJntPos :=m_caliPlanner[m_caliTrajIdx].evaluate(m_timePeriod, jntPos=> m_cmdJntPos, jntVel=>m_cmdJntVel, jntAcc=> m_cmdJntAcc);

// check if to transit to next segment
curJntVel :=i_slaveArm.curJntVel;
IF(m_timePeriod > m_caliPlanner[m_caliTrajIdx].duration  AND norm(curJntVel)<7*GVL_SlaveControlParameters.g_jntStaticVelThres) THEN
	m_caliTrajIdx:=m_caliTrajIdx+1;
	m_timePeriod:=0;
END_IF

// check if to terminated
IF(m_caliTrajIdx > m_caliMotionSegs) THEN
	m_isFinished:=TRUE;
END_IF
END_METHOD

METHOD PUBLIC init : BOOL
VAR_IN_OUT CONSTANT
	i_slaveArm	:FB_SlaveArm;
END_VAR
VAR_IN_OUT 
	r_slaveArmCtrlCmd :ST_SlaveArmCtrlCmds;
END_VAR

VAR
	i,j :INT;
	initJntPos,startJntPos,endJntPos :Vec8d;

END_VAR
SUPER^.Init(i_slaveArm,r_slaveArmCtrlCmd);
m_caliTrajIdx :=1;
m_jntOPMode := g_slaveAllPosTrqMode;

// traj plan
// fisrt segment
initJntPos:=i_slaveArm.curJntPos;
startJntPos:=initJntPos;
endJntPos:=startJntPos;
FOR j:=1 TO 3 DO 
	endJntPos[j]:=m_graCaliTraj[1,j];
END_FOR
m_caliPlanner[1].init(startJntPos,endJntPos,m_caliMaxjntVel, m_caliMaxJntAcc, m_caliMaxJntJerk);

// other segments
FOR i:=2 TO m_caliMotionSegs DO 
	startJntPos := endJntPos;
	endJntPos:=startJntPos;
	FOR j:=1 TO 3 DO 
		endJntPos[j]:=m_graCaliTraj[i,j];
	END_FOR
	m_caliPlanner[i].init(startJntPos,endJntPos,m_caliMaxjntVel, m_caliMaxJntAcc, m_caliMaxJntJerk);
END_FOR

// update commands to arm
copyCmds(r_slaveArmCtrlCmd);
END_METHOD

END_FUNCTION_BLOCK

// ---- Mains/CartControl.TcPOU
PROGRAM CartControl
VAR
	// cart instance
	m_cartRobot :FB_CartRobot;
	
	// Output cart status
	m_cartStatus AT%Q* : ST_CartStatus;
	
	
	m_cartDataPool: ST_CartInputDataPool;
	
	// wait time before cart init for ethercat to be statble 
	m_cartInitWaitTime : LREAL:=0;
	
	// cart init flag
	m_cartInit :BOOL :=FALSE;
	
	m_workHeartTon0 : TON;
	m_workHeartTon1 : TON;
	m_dumpEnergy : UINT:=51;
	m_cartInSterileStateTon :Ton;
	m_cartInSterileState :BOOL;
	//Aseptic sleeve is installed flag
	m_asepticInstalledFlag : Vec4b;
	m_slaveArmDisableFlag : Vec4b;
END_VAR

// wait communication to be stable
IF(m_cartInitWaitTime<g_robotInitWaitTime) THEN
	m_cartInitWaitTime := m_cartInitWaitTime+g_cartCtrlCycleTime;
	RETURN;
END_IF

// cart init
IF m_cartInit =FALSE THEN
	m_cartRobot.Init();
	m_cartInit:=TRUE;
END_IF

// input from UI
UIInputProcess();

//Aseptic sleeve deployment completed
m_cartDataPool.m_cartStatus.m_asepticDeployCompletedFlag := SlaveArmControl.m_slaveRobot.m_panelMountedFlag[1] AND SlaveArmControl.m_slaveRobot.m_panelMountedFlag[2]
																									AND SlaveArmControl.m_slaveRobot.m_panelMountedFlag[3] AND SlaveArmControl.m_slaveRobot.m_panelMountedFlag[4];

// cart run
m_cartRobot.run(m_cartDataPool);


UIOutputProcess();

// tranform data from UI(global variable write by ADS) to ST_UIData
METHOD UIInputProcess : BOOL
VAR_INPUT
END_VAR
VAR
	i:int;
END_VAR
// cart Joystick data
m_cartDataPool.m_UIData.m_joystickDataFromUI := GVL_com_upper_PC.a8usb_rec_array;

m_cartDataPool.m_UIData.m_ctrlEnableFromUI := GVL_com_upper_PC.ui_control;

//limit_height:UINT;  上位机的高度值单位是mm，系统的高度值单位是m，底座高度是1850mm
//打开ui_control.limit_height_adjusting后可以调整立柱，并实时将立柱当前高度上传
IF (GVL_com_upper_PC.ui_control.limit_height_adjusting=TRUE) THEN
	m_cartDataPool.m_UIData.m_standColumnHightLimit := GVL_CartMotorParameters.g_maxJntPos[5];
	GVL_com_upper_PC.limit_height :=LREAL_TO_UINT (m_cartRobot.m_slaveCart.curJntPos[5] * 1000 + 1850);
ELSIF 	 (GVL_com_upper_PC.ui_control.limit_height_adjusting=FALSE) AND GVL_com_upper_PC.enable_limit_height AND ABS((m_cartDataPool.m_UIData.m_standColumnHightLimit *1000+1850)-GVL_com_upper_PC.limit_height)>5 THEN
	m_cartDataPool.m_UIData.m_standColumnHightLimit := UINT_TO_LREAL(GVL_com_upper_PC.limit_height-1850)/1000;
ELSIF GVL_com_upper_PC.enable_limit_height=FALSE THEN
	m_cartDataPool.m_UIData.m_standColumnHightLimit := GVL_CartMotorParameters.g_maxJntPos[5];
END_IF


//Surgical orientation selection
m_cartDataPool.m_UIData.m_surgicalSite := GVL_com_upper_PC.surgical_site;
m_cartDataPool.m_UIData.m_surgicalLocation := GVL_com_upper_PC.surgical_location;

m_dumpEnergy := GVL_com_upper_PC.battery_power_value;
END_METHOD

METHOD UIOutputProcess : BOOL
VAR_INPUT
END_VAR
VAR 
	i : INT;
END_VAR
//TODO
//work heart
m_workHeartTon0(IN:= GVL_com_upper_PC.work_heart = 1, PT:= T#1S, Q=> , ET=> );
m_workHeartTon1(IN:= GVL_com_upper_PC.work_heart = 0, PT:= T#1S, Q=> , ET=> );
IF m_workHeartTon0.Q THEN
	GVL_com_upper_PC.work_heart :=0 ;
ELSIF m_workHeartTon1.Q THEN
	GVL_com_upper_PC.work_heart  :=1 ;
END_IF

GVL_com_upper_PC.cart_operation.draping_posture_state := m_cartRobot.m_slaveCart.m_cartDataFromUI.m_cartDrapingState;
GVL_com_upper_PC.cart_operation.docking_posture_state := m_cartRobot.m_slaveCart.m_cartDataFromUI.m_cartDockingState;

GVL_com_upper_PC.torcars_status := INT_TO_BOOL(m_cartRobot.m_slaveCart.m_trocarOnFlag);

GVL_com_upper_PC.Cart_running_alone := NOT SlaveArmControl.m_slaveRobot.m_masterOnLine;
GVL_com_upper_PC.has_Cart_recoverable_error := 0;

IF GVL_com_upper_PC.surgical_status = 1 THEN
	IF m_cartDataPool.m_cartStatus.m_asepticDeployCompletedFlag =FALSE THEN
		m_slaveArmDisableFlag := g_zeroVec4b;
	END_IF
ELSE
	m_slaveArmDisableFlag := SlaveArmControl.m_slaveInputDataPool.m_UIData.m_slaveArmDisableFlag;	
END_IF

FOR i := 1 TO 4 BY 1 DO
	m_asepticInstalledFlag[i] := m_slaveArmDisableFlag[i] OR SlaveArmControl.m_slaveRobot.m_panelMountedFlag[i];
END_FOR

GVL_com_upper_PC.Cart_operation.Arm1_setup_sterile_state := BOOL_TO_UINT(m_asepticInstalledFlag[1]); 
GVL_com_upper_PC.Cart_operation.Arm2_setup_sterile_state := BOOL_TO_UINT(m_asepticInstalledFlag[2]); 
GVL_com_upper_PC.Cart_operation.Arm3_setup_sterile_state := BOOL_TO_UINT(m_asepticInstalledFlag[3]); 
GVL_com_upper_PC.Cart_operation.Arm4_setup_sterile_state := BOOL_TO_UINT(m_asepticInstalledFlag[4]); 

GVL_com_upper_PC.Cart_operation.setup_sterile_state := BOOL_TO_UINT(m_asepticInstalledFlag[1]) AND BOOL_TO_UINT(m_asepticInstalledFlag[2]) AND BOOL_TO_UINT(m_asepticInstalledFlag[3]) AND BOOL_TO_UINT(m_asepticInstalledFlag[4]) ;

GVL_com_upper_PC.Cart_operation.scope_install_state := BOOL_TO_UINT(SlaveArmControl.m_slaveRobot.m_endoscopeMounted);

FOR i := 1 TO 4 BY 1 DO
	IF NOT SlaveArmControl.m_slaveRobot.m_slaveArms[i].instrument.onChipData.m_Instrutype=InstruType_endoscope THEN
		IF SlaveArmControl.m_slaveRobot.m_instrumentMountedFlag[i] AND SlaveArmControl.m_slaveRobot.m_endoscopeMounted THEN
			GVL_com_upper_PC.Cart_operation.all_fixed_point_confirm := 1;
			EXIT;
		ELSE
			GVL_com_upper_PC.Cart_operation.all_fixed_point_confirm := 0;
		END_IF	
	END_IF	
END_FOR


//Cart_static_in_sterile_state:UINT; //台车进入无菌区，并且台车停止运动(连续10s没有运动)，0：没有完成，1：完成
IF m_cartRobot.m_slaveCart.m_cartDataFromUI.m_cartDockingState = 1 THEN
	IF m_cartRobot.m_CartState = CartJointState_Movement THEN
		m_cartInSterileState := FALSE;
	ELSIF m_cartRobot.m_lastCartState = CartJointState_Movement THEN
		m_cartInSterileState := TRUE;
	END_IF
ELSE
	m_cartInSterileState := FALSE;
	GVL_com_upper_PC.Cart_operation.Cart_static_in_sterile_state:=0;
END_IF
m_cartInSterileStateTon(IN:= m_cartInSterileState, PT:= T#10S, Q=> , ET=> );
IF m_cartInSterileStateTon.Q THEN
	GVL_com_upper_PC.Cart_operation.Cart_static_in_sterile_state:=1;
END_IF

GVL_com_upper_PC.manual_mode := NOT m_cartRobot.m_slaveCart.m_stabilizFootSensorManual;
END_METHOD

END_PROGRAM

// ---- Mains/SafetyCheck.TcPOU
PROGRAM SafetyCheck
VAR
	// slave robot information, including arm status and cartesian data
	m_slaveStatus AT %I* :ST_slaveStatus;
	
	// slave robot joint data
	m_slaveJointData AT %I* :ST_slaveJointData;
	
	// setup robot information
	m_setupStatus AT %I* :ST_SetupStatus;
	
	// setup robot joint data
	m_setupJointsData AT %I* :ST_SetupJointData;
	
	// error check result
	m_safetyCheckData AT %Q* :ST_SafetyData;
	
	m_initFlag:bool;
	m_cartCheck :FB_CartCheck;
	m_setupArmCheck:FB_SetupArmCheck;
	m_slaveArmCheck:FB_SlaveArmCheck;
	
	i: INT;
END_VAR

// reset data
IF FALSE = m_initFlag  THEN
	FOR i:=1  TO g_sArmNum DO 
		m_safetyCheckData.m_slaveErrFlag[i]:=FALSE;
		m_safetyCheckData.m_setupErrFlag[i]:=FALSE;
		m_safetyCheckData.m_cartErrFlag:=false;
	END_FOR
	m_initFlag:=TRUE;
END_IF

m_slaveArmCheck.check(m_slaveStatus,m_slaveJointData, o_errorFlag=>m_safetyCheckData.m_slaveErrFlag);
m_setupArmCheck.check(m_setupStatus,m_setupJointsData, o_errorFlag=>m_safetyCheckData.m_setupErrFlag);

END_PROGRAM

// ---- SafetyCheck/FB_SetupArmCheck.TcPOU
FUNCTION_BLOCK FB_SetupArmCheck
VAR_INPUT
END_VAR
VAR_OUTPUT
END_VAR
VAR
	// final arm error flag
	m_armErrFlag :ARRAY[1..g_sArmNum] OF BOOL:=[4(FALSE)];
	
	// original position of remote center point when fisrt enter hold state
	m_dsrRcpPos :ARRAY[1..g_sArmNum] OF Vec3d;
	
	// rcp error flag
	m_rcpPosErrFlag :ARRAY[1..g_sArmNum] OF BOOL;
	m_rcpPosErrCounts :ARRAY[1..g_sArmNum] OF INT := [4(0)];
	m_rcpPosErr :ARRAY[1..g_sArmNum] OF Vec3d;		// rcp position error
	
	// joint control error flag
	m_jntCtrlErrFlag :ARRAY[1..g_sArmNum] OF Vec5b;
	m_jntCtrlErrCounts :ARRAY[1..g_sArmNum] OF Vec5i;
	m_jntCtrlErr:ARRAY[1..g_sArmNum]  OF Vec5d;	// joint position control error
	
	// joint encoder error flag
	m_jntEncErrFlag :ARRAY[1..g_sArmNum] OF Vec5b;
	m_jntEncErrCounts :ARRAY[1..g_sArmNum] OF Vec5i ;
	m_jntEncErr:ARRAY[1..g_sArmNum]  OF Vec5d;		// motor and joint encoder error
	
	// joint velocity error flag
	m_jntVelErrFlag :ARRAY[1..g_sArmNum] OF Vec5b;
	m_jntVelErrCounts :ARRAY[1..g_sArmNum] OF Vec5i ;
	
	// joint position limit error flag
	m_jntLimitErrFlag :ARRAY[1..g_sArmNum] OF Vec5b;
	m_jntLimitErrCounts :ARRAY[1..g_sArmNum] OF Vec5i;
	

END_VAR

METHOD check : BOOL
VAR_IN_OUT CONSTANT
	i_setupStatus : ST_SetupStatus;
	i_setupJointData :ST_SetupJointData;
END_VAR
VAR_OUTPUT
	o_errorFlag :ARRAY[1..g_sArmNum] OF BOOL ;
END_VAR

VAR
	i ,j:INT ;
END_VAR
// calculate error
FOR i:=1 TO g_sArmNum DO 
	// update rcp
	IF i_setupStatus.m_armState[i] <> SetupArmState_Hold THEN
		m_dsrRcpPos[i] := i_setupStatus.m_rcPos[i];
	END_IF

	// stop check if arm is already in error state
	IF m_armErrFlag[i] OR i_setupStatus.m_armState[i] = SetupArmState_Error THEN 
		CONTINUE;
	END_IF
	
	// only check rcp when slave in master-slave control state (for master-slave control)
	m_rcpPosErrFlag[i]:=FALSE;
	IF SlaveArmControl.m_slaveStatus.m_armState[i] = SlaveArmState_MasterSlave THEN 
		m_rcpPosErrFlag[i]:=rcpErrCheck(m_dsrRcpPos[i],  i_setupStatus.m_rcPos[i], m_rcpPosErrCounts[i] ,m_rcpPosErr[i]);
	END_IF
	
	// joint control error
	m_jntCtrlErrFlag[i]:=jntCtrlErrCheck(i_setupJointData.m_cmdJntPos[i], i_setupJointData.m_curJntPos[i],
										m_jntCtrlErrCounts[i], m_jntCtrlErr[i]);
	
	// encoder error
	m_jntEncErrFlag[i]:=jntEncErrCheck(i_setupJointData.m_curMotorPos[i], i_setupJointData.m_curLinkPos[i],
										m_jntEncErrCounts[i] , m_jntEncErr[i]);
							
	// joint limit error
	m_jntLimitErrFlag[i]:=jntLimitErrCheck(i, i_setupJointData.m_curJntPos[i],m_jntLimitErrCounts[i]);
										
	// final arm error status check
	IF  m_rcpPosErrFlag[i] THEN
		m_armErrFlag[i]:=TRUE;
		CONTINUE;
	END_IF
	
	FOR j:=1 TO g_setupJntNum DO 
		IF  m_jntCtrlErrFlag[i][j] OR m_jntEncErrFlag[i][j] OR m_jntVelErrFlag[i][j] OR m_jntLimitErrFlag[i][j]  THEN
			m_armErrFlag[i]:=TRUE;
			EXIT;
		END_IF
	END_FOR
	
END_FOR

o_errorFlag:=m_armErrFlag;
END_METHOD

METHOD jntCtrlErrCheck : Vec5b
VAR_INput
	i_cmdJntPos : Vec5d;
	i_curJntPos : Vec5d;
END_VAR
VAR_IN_OUT
	r_errCount:Vec5i;
	r_jntCtrlErr :Vec5d;
END_VAR

VAR
	i :INT;
	err:Vec5d;
END_VAR
vecSub(i_cmdJntPos,i_curJntPos,  err);
r_jntCtrlErr:=err;

// joint error check
FOR i:=1 TO g_setupJntNum DO 
	IF ABS(r_jntCtrlErr[i]) > g_setupMaxJntCtrlErr[i] THEN
		r_errCount[i]:=r_errCount[i]+1;
	ELSE
		r_errCount[i] :=0;
	END_IF
	jntCtrlErrCheck[i]:= r_errCount[i]>=g_faultTriggerCounts;
END_FOR
END_METHOD

METHOD jntEncErrCheck : Vec5b
VAR_INput
	i_motorJntPos : Vec5d;
	i_linkJntPos : Vec5d;
END_VAR
VAR_IN_OUT
	r_errCount:Vec5i;
	r_jntEncErr :Vec5d;
END_VAR

VAR
	i :INT;
	err : vec5d;
END_VAR
vecSub(i_motorJntPos,i_linkJntPos,  err);
r_jntEncErr:=err;

// joint error check
FOR i:=1 TO g_setupJntNum DO 
	IF  ABS(r_jntEncErr[i]) > g_setupMaxJntCtrlErr[i] THEN
		r_errCount[i]:=r_errCount[i]+1;
	ELSE
		r_errCount[i] :=0;
	END_IF
	jntEncErrCheck[i]:= r_errCount[i]>=g_faultTriggerCounts;
END_FOR
END_METHOD

METHOD jntLimitErrCheck : Vec5b
VAR_INPUT
	i_armIdx : INT;
	i_curJntPos : Vec5d;
END_VAR
VAR_IN_OUT
	r_errCount:Vec5i;
END_VAR

VAR
	i :INT;
END_VAR
// joint limit check
FOR i:=1 TO 5 DO 
	IF  i_curJntPos[i] > GVL_SetupMotorParameters.g_maxJntPos[i_armIdx,i] + g_setupJntPosLimitBuffer[i] OR
		i_curJntPos[i] < GVL_SetupMotorParameters.g_minJntPos[i_armIdx,i] - g_setupJntPosLimitBuffer[i] THEN
		r_errCount[i]:=r_errCount[i]+1;
	ELSE
		r_errCount[i] :=0;	
	END_IF
	jntLimitErrCheck[i]:= r_errCount[i]>=g_faultTriggerCounts;
END_FOR
END_METHOD

METHOD rcpErrCheck : BOOL
VAR_INPUT
	i_cmdPos : Vec3d;
	i_curPos : Vec3d;
END_VAR
VAR_IN_OUT
	r_errCount:INT;
	r_posErr :Vec3d;
END_VAR

VAR
	err:Vec3d;
END_VAR
vecSub(i_cmdPos, i_curPos,err);
r_posErr:=err;

IF  (norm(err)>g_rcpDeviationThres) THEN
	r_errCount:= r_errCount +1;
ELSE 
	r_errCount:=0;
END_IF
rcpErrCheck := r_errCount >= g_faultTriggerCounts;
END_METHOD

END_FUNCTION_BLOCK
